// Mitsubishi GX Works2 project: 아날로그속도제어   PLC: Q03UDV

PROGRAM MAIN
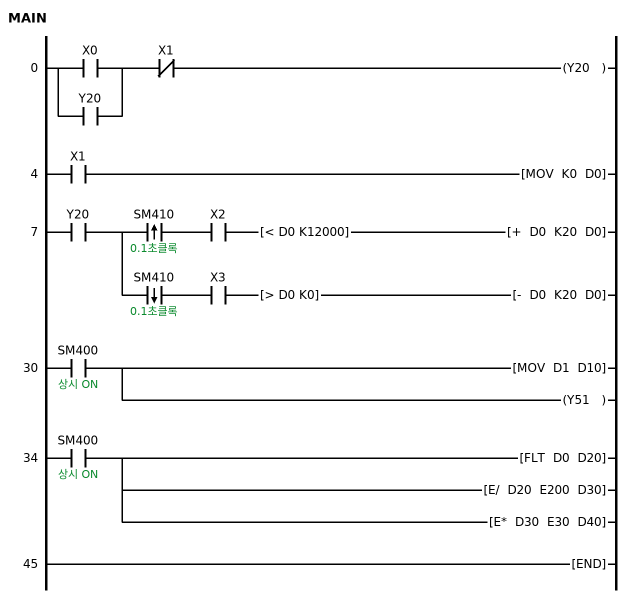
0     LD      X0
      OR      Y20
      ANI     X1
      OUT     Y20
4     LD      X1
      MOV     K0 D0
7     LD      Y20
      MPS
      ANDP    SM410  ; 0.1초클록
      AND     X2
      AND<    D0 K12000
      +       D0 K20 D0
      MPP
      ANDF    SM410  ; 0.1초클록
      AND     X3
      AND>    D0 K0
      -       D0 K20 D0
30    LD      SM400  ; 상시 ON
      MOV     D1 D10
      OUT     Y51
34    LD      SM400  ; 상시 ON
      FLT     D0 D20
      E/      D20 E200 D30
      E*      D30 E30 D40
45    END
END_PROGRAM
